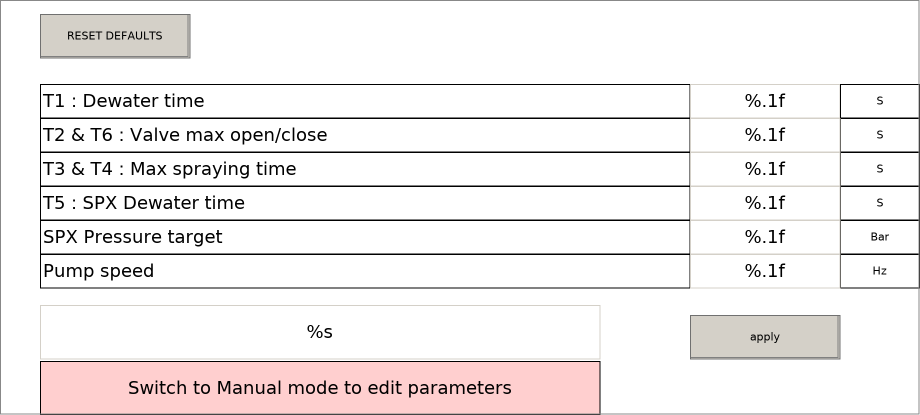
VISUALIZATION visu_Params  // 920x415
    Rectangle (40,84 650x34), "T1 : Dewater time"
    Textfield (690,84 150x34), "%.1f", text variable: PRG_Params.rEditDewater_s, input disabled if: NOT PRG_Spray.bManualActive
        OnMouseClick: write the text variable via VisuDialogs.Numpad, min 0, max 9999999
    Rectangle (840,84 80x34), "S"
    Rectangle (840,118 80x34), "S"
    Rectangle (40,118 650x34), "T2 & T6 : Valve max open/close"
    Textfield (690,118 150x34), "%.1f", text variable: PRG_Params.rEditValveMax_s, input disabled if: NOT PRG_Spray.bManualActive
        OnMouseClick: write the text variable via VisuDialogs.Numpad, min 0, max 9999999
    Rectangle (840,152 80x34), "S"
    Rectangle (40,152 650x34), "T3 & T4 : Max spraying time"
    Textfield (690,152 150x34), "%.1f", text variable: PRG_Params.rEditSprayTime_s, input disabled if: NOT PRG_Spray.bManualActive
        OnMouseClick: write the text variable via VisuDialogs.Numpad, min 0, max 9999999
    Rectangle (840,186 80x34), "S"
    Rectangle (40,186 650x34), "T5 : SPX Dewater time"
    Textfield (690,186 150x34), "%.1f", text variable: PRG_Params.rEditSPXDewater_s, input disabled if: NOT PRG_Spray.bManualActive
        OnMouseClick: write the text variable via VisuDialogs.Numpad, min 0, max 9999999
    Rectangle (840,220 80x34), "Bar"
    Rectangle (40,220 650x34), "SPX Pressure target"
    Textfield (690,220 150x34), "%.1f", text variable: PRG_Params.rEditPressTarget, input disabled if: NOT PRG_Spray.bManualActive
        OnMouseClick: write the text variable via VisuDialogs.Numpad, min 0, max 9999999
    Rectangle (840,254 80x34), "Hz"
    Rectangle (40,254 650x34), "Pump speed"
    Textfield (690,254 150x34), "%.1f", text variable: PRG_Params.rEditPumpSpeed, input disabled if: NOT PRG_Spray.bManualActive
        OnMouseClick: write the text variable via VisuDialogs.Numpad, min 0, max 9999999
    Button (690,315 150x44), "apply", input disabled if: NOT PRG_Spray.bManualActive
        tap PRG_Params.bBtnApply
    Textfield (40,305 560x54), "%s", text variable: PRG_Params.sParamStatus, invisible if: NOT PRG_Params.bMsgVisible
    Rectangle (40,361 560x54), "Switch to Manual mode to edit parameters", invisible if: NOT (PRG_Params.bMsgVisible AND NOT PRG_Spray.bManualActive)
    Button (40,14 150x44), "RESET DEFAULTS", input disabled if: NOT PRG_Spray.bManualActive
        tap PRG_Params.bBtnReset
END_VISUALIZATION

(* stored: Version 1.1.0.1, ProductVersion 3.1.4026.18
   Visu visu_Params: Id {d1b07259-a55d-40ff-ab2b-41f79a124630} *)
